// TIA Portal V17 export
// export: Created 2025-03-07T09:17:01.8029141Z, ExportSetting WithDefaults, DisplayName Totally Integrated Automation Portal, DisplayVersion V17 Update 8, DisplayName TIA Portal Openness, DisplayVersion V17 Update 8, DisplayName TIA Portal Version Control Interface, DisplayVersion V17, DisplayName SINAMICS Startdrive Advanced, DisplayVersion V17 SP2, DisplayName SINAMICS Startdrive G110M, G120, G120C, G120D, G120P, G115D, DisplayVersion V17 SP2, DisplayName SINAMICS Startdrive G130, G150, S120, S150, SINAMICS MV, S210, DisplayVersion V17 SP2, DisplayName STEP 7 Professional, DisplayVersion V17 Update 8, DisplayName SINUMERIK ONE STEP 7 Toolbox, DisplayVersion V17 Update 12, DisplayName SINUMERIK 840D sl STEP 7 Toolbox, DisplayVersion V17 Update 12, DisplayName STEP 7 Safety, DisplayVersion V17 Update 6, DisplayName WinCC Advanced, DisplayVersion V17 Update 8
FUNCTION "FC7341_POWDER_PLC_TO_MACHINE_INTERLOCK" : Void   // FC7341, LAD
{ S7_Optimized_Access := 'TRUE' }
VERSION : 0.1
// stored: AutoNumber false, IsIECCheckEnabled false, SetENOAutomatically false, UDAEnableTagReadback false
   VAR_TEMP
      COUNT_FOR_ERROR : Int;
      RET_VAL_1 : Int;
   END_VAR
   VAR CONSTANT
      FC_NUMBER : DInt := 7341;
   END_VAR
BEGIN

REGION Network 1: LIFE BIT
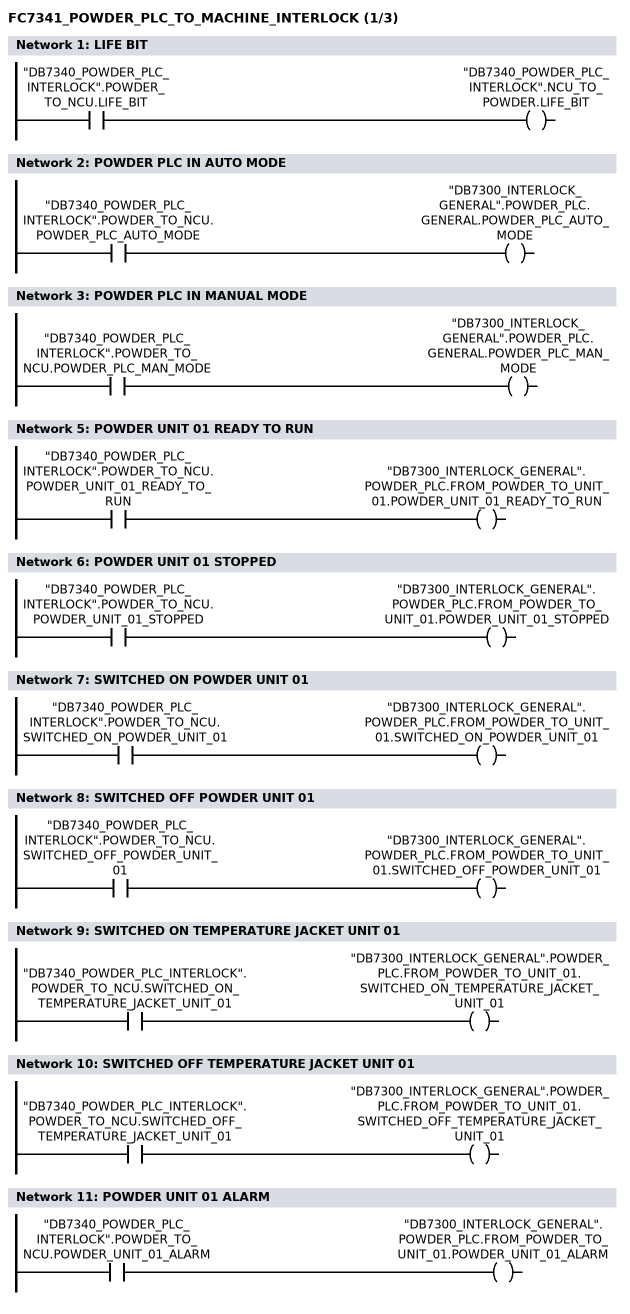
   RUNG wire#powerrail
      Contact( "DB7340_POWDER_PLC_INTERLOCK".POWDER_TO_NCU.LIFE_BIT )
      Coil( "DB7340_POWDER_PLC_INTERLOCK".NCU_TO_POWDER.LIFE_BIT )
   END_RUNG
   // the same network as SCL:
   "DB7340_POWDER_PLC_INTERLOCK".NCU_TO_POWDER.LIFE_BIT := "DB7340_POWDER_PLC_INTERLOCK".POWDER_TO_NCU.LIFE_BIT;
END_REGION

REGION Network 2: POWDER PLC IN AUTO MODE
   RUNG wire#powerrail
      Contact( "DB7340_POWDER_PLC_INTERLOCK".POWDER_TO_NCU.POWDER_PLC_AUTO_MODE )
      Coil( "DB7300_INTERLOCK_GENERAL".POWDER_PLC.GENERAL.POWDER_PLC_AUTO_MODE )
   END_RUNG
   // the same network as SCL:
   "DB7300_INTERLOCK_GENERAL".POWDER_PLC.GENERAL.POWDER_PLC_AUTO_MODE := "DB7340_POWDER_PLC_INTERLOCK".POWDER_TO_NCU.POWDER_PLC_AUTO_MODE;
END_REGION

REGION Network 3: POWDER PLC IN MANUAL MODE
   RUNG wire#powerrail
      Contact( "DB7340_POWDER_PLC_INTERLOCK".POWDER_TO_NCU.POWDER_PLC_MAN_MODE )
      Coil( "DB7300_INTERLOCK_GENERAL".POWDER_PLC.GENERAL.POWDER_PLC_MAN_MODE )
   END_RUNG
   // the same network as SCL:
   "DB7300_INTERLOCK_GENERAL".POWDER_PLC.GENERAL.POWDER_PLC_MAN_MODE := "DB7340_POWDER_PLC_INTERLOCK".POWDER_TO_NCU.POWDER_PLC_MAN_MODE;
END_REGION

REGION Network 4: //////////_UNIT_01_//////////
END_REGION

REGION Network 5: POWDER UNIT 01 READY TO RUN
   RUNG wire#powerrail
      Contact( "DB7340_POWDER_PLC_INTERLOCK".POWDER_TO_NCU.POWDER_UNIT_01_READY_TO_RUN )
      Coil( "DB7300_INTERLOCK_GENERAL".POWDER_PLC.FROM_POWDER_TO_UNIT_01.POWDER_UNIT_01_READY_TO_RUN )
   END_RUNG
   // the same network as SCL:
   "DB7300_INTERLOCK_GENERAL".POWDER_PLC.FROM_POWDER_TO_UNIT_01.POWDER_UNIT_01_READY_TO_RUN := "DB7340_POWDER_PLC_INTERLOCK".POWDER_TO_NCU.POWDER_UNIT_01_READY_TO_RUN;
END_REGION

REGION Network 6: POWDER UNIT 01 STOPPED
   RUNG wire#powerrail
      Contact( "DB7340_POWDER_PLC_INTERLOCK".POWDER_TO_NCU.POWDER_UNIT_01_STOPPED )
      Coil( "DB7300_INTERLOCK_GENERAL".POWDER_PLC.FROM_POWDER_TO_UNIT_01.POWDER_UNIT_01_STOPPED )
   END_RUNG
   // the same network as SCL:
   "DB7300_INTERLOCK_GENERAL".POWDER_PLC.FROM_POWDER_TO_UNIT_01.POWDER_UNIT_01_STOPPED := "DB7340_POWDER_PLC_INTERLOCK".POWDER_TO_NCU.POWDER_UNIT_01_STOPPED;
END_REGION

REGION Network 7: SWITCHED ON POWDER UNIT 01
   RUNG wire#powerrail
      Contact( "DB7340_POWDER_PLC_INTERLOCK".POWDER_TO_NCU.SWITCHED_ON_POWDER_UNIT_01 )
      Coil( "DB7300_INTERLOCK_GENERAL".POWDER_PLC.FROM_POWDER_TO_UNIT_01.SWITCHED_ON_POWDER_UNIT_01 )
   END_RUNG
   // the same network as SCL:
   "DB7300_INTERLOCK_GENERAL".POWDER_PLC.FROM_POWDER_TO_UNIT_01.SWITCHED_ON_POWDER_UNIT_01 := "DB7340_POWDER_PLC_INTERLOCK".POWDER_TO_NCU.SWITCHED_ON_POWDER_UNIT_01;
END_REGION

REGION Network 8: SWITCHED OFF POWDER UNIT 01
   RUNG wire#powerrail
      Contact( "DB7340_POWDER_PLC_INTERLOCK".POWDER_TO_NCU.SWITCHED_OFF_POWDER_UNIT_01 )
      Coil( "DB7300_INTERLOCK_GENERAL".POWDER_PLC.FROM_POWDER_TO_UNIT_01.SWITCHED_OFF_POWDER_UNIT_01 )
   END_RUNG
   // the same network as SCL:
   "DB7300_INTERLOCK_GENERAL".POWDER_PLC.FROM_POWDER_TO_UNIT_01.SWITCHED_OFF_POWDER_UNIT_01 := "DB7340_POWDER_PLC_INTERLOCK".POWDER_TO_NCU.SWITCHED_OFF_POWDER_UNIT_01;
END_REGION

REGION Network 9: SWITCHED ON TEMPERATURE JACKET UNIT 01
   RUNG wire#powerrail
      Contact( "DB7340_POWDER_PLC_INTERLOCK".POWDER_TO_NCU.SWITCHED_ON_TEMPERATURE_JACKET_UNIT_01 )
      Coil( "DB7300_INTERLOCK_GENERAL".POWDER_PLC.FROM_POWDER_TO_UNIT_01.SWITCHED_ON_TEMPERATURE_JACKET_UNIT_01 )
   END_RUNG
   // the same network as SCL:
   "DB7300_INTERLOCK_GENERAL".POWDER_PLC.FROM_POWDER_TO_UNIT_01.SWITCHED_ON_TEMPERATURE_JACKET_UNIT_01 := "DB7340_POWDER_PLC_INTERLOCK".POWDER_TO_NCU.SWITCHED_ON_TEMPERATURE_JACKET_UNIT_01;
END_REGION

REGION Network 10: SWITCHED OFF TEMPERATURE JACKET UNIT 01
   RUNG wire#powerrail
      Contact( "DB7340_POWDER_PLC_INTERLOCK".POWDER_TO_NCU.SWITCHED_OFF_TEMPERATURE_JACKET_UNIT_01 )
      Coil( "DB7300_INTERLOCK_GENERAL".POWDER_PLC.FROM_POWDER_TO_UNIT_01.SWITCHED_OFF_TEMPERATURE_JACKET_UNIT_01 )
   END_RUNG
   // the same network as SCL:
   "DB7300_INTERLOCK_GENERAL".POWDER_PLC.FROM_POWDER_TO_UNIT_01.SWITCHED_OFF_TEMPERATURE_JACKET_UNIT_01 := "DB7340_POWDER_PLC_INTERLOCK".POWDER_TO_NCU.SWITCHED_OFF_TEMPERATURE_JACKET_UNIT_01;
END_REGION

REGION Network 11: POWDER UNIT 01 ALARM
   RUNG wire#powerrail
      Contact( "DB7340_POWDER_PLC_INTERLOCK".POWDER_TO_NCU.POWDER_UNIT_01_ALARM )
      Coil( "DB7300_INTERLOCK_GENERAL".POWDER_PLC.FROM_POWDER_TO_UNIT_01.POWDER_UNIT_01_ALARM )
   END_RUNG
   // the same network as SCL:
   "DB7300_INTERLOCK_GENERAL".POWDER_PLC.FROM_POWDER_TO_UNIT_01.POWDER_UNIT_01_ALARM := "DB7340_POWDER_PLC_INTERLOCK".POWDER_TO_NCU.POWDER_UNIT_01_ALARM;
END_REGION

REGION Network 12: POWDER FEEDER 1 ACTUAL VALUES
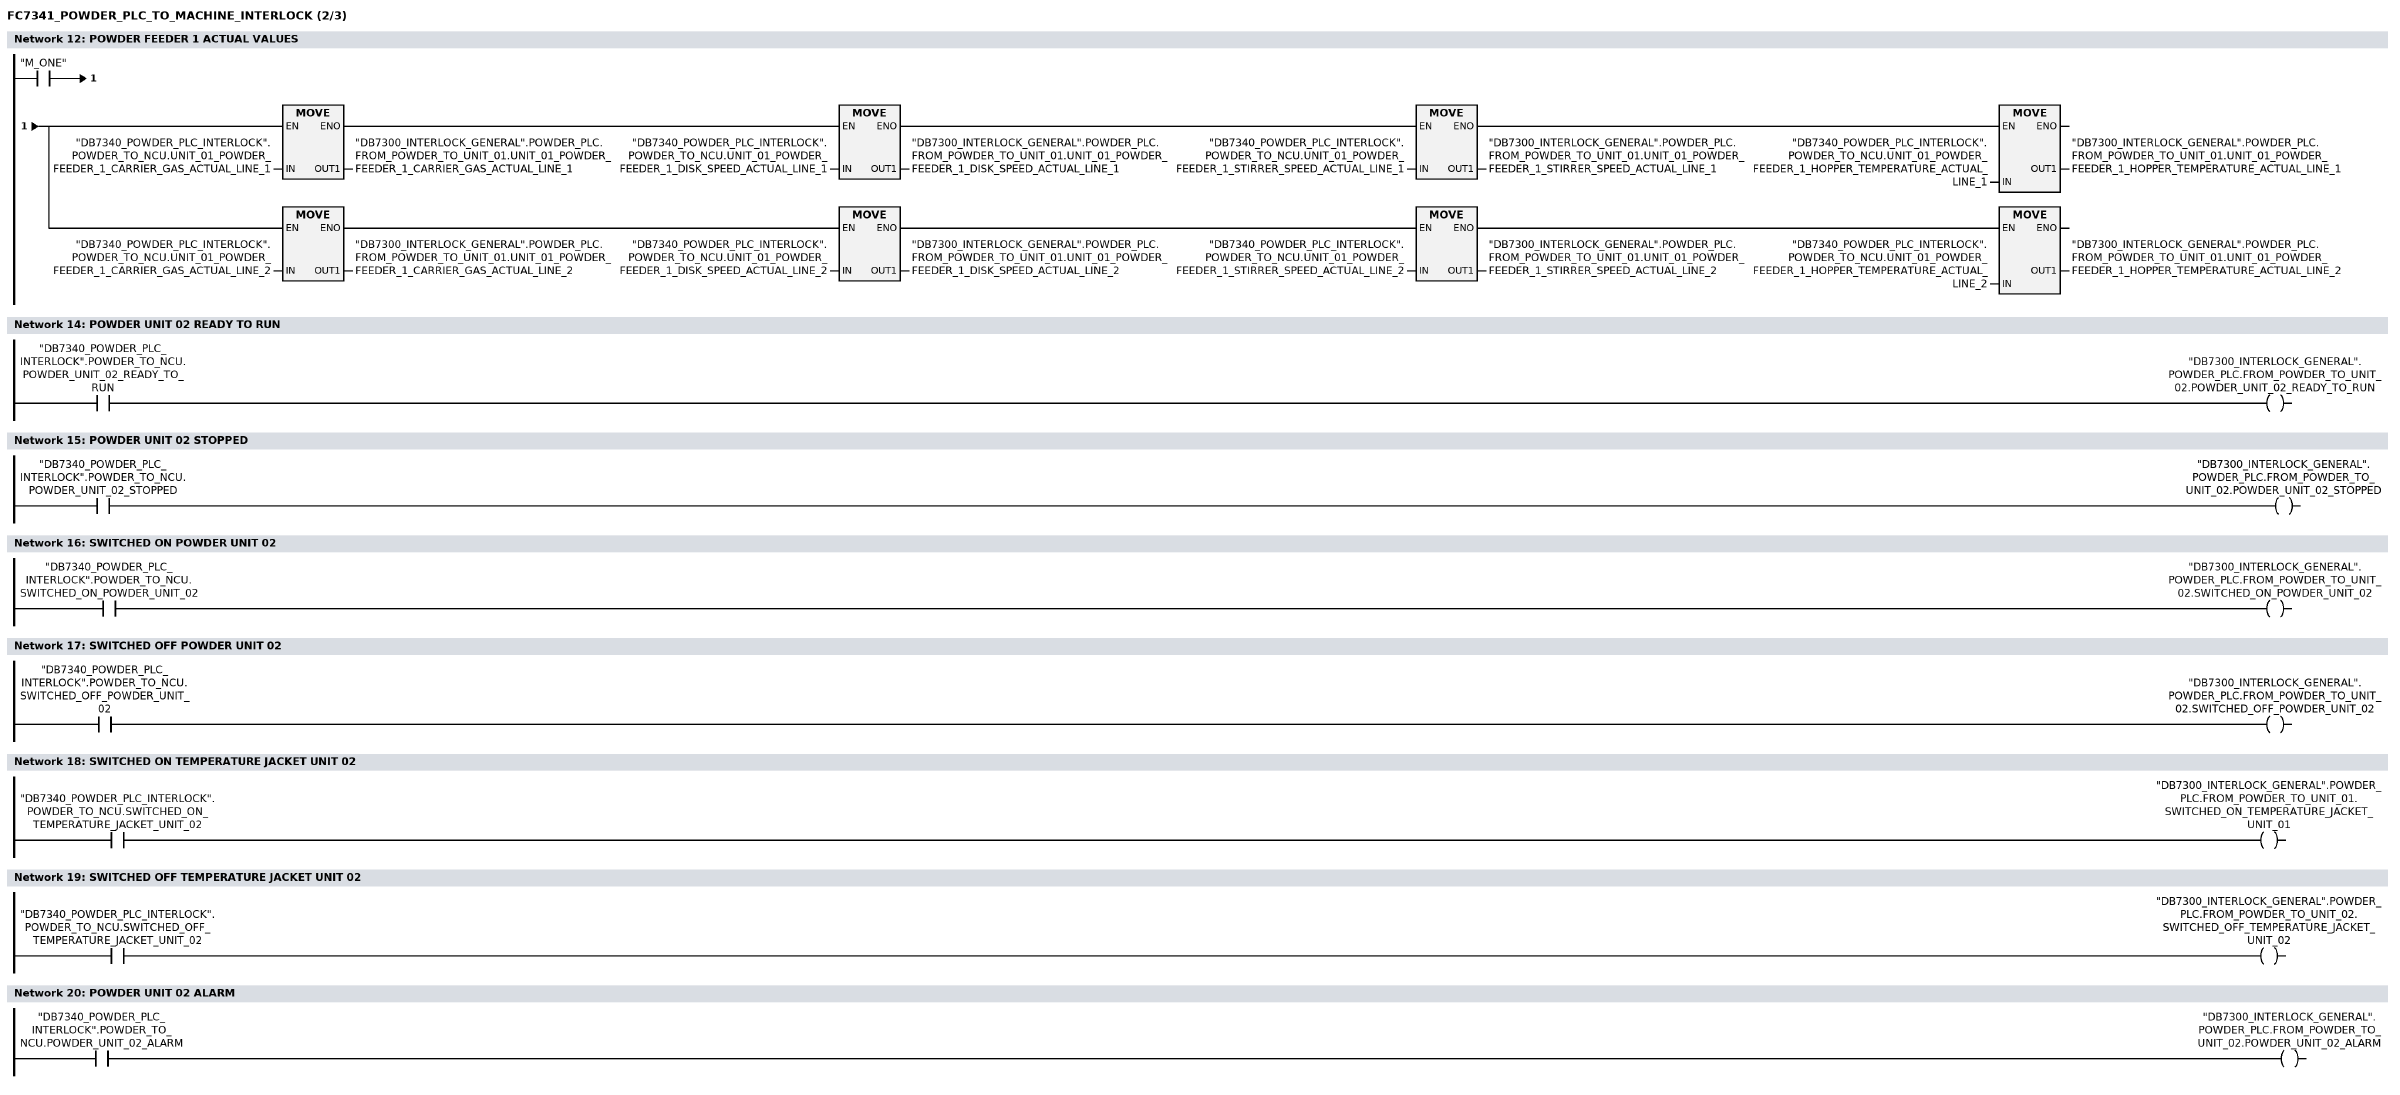
   RUNG wire#powerrail
      Contact( "M_ONE" )
      wire#w1
      Move(in := "DB7340_POWDER_PLC_INTERLOCK".POWDER_TO_NCU.UNIT_01_POWDER_FEEDER_1_CARRIER_GAS_ACTUAL_LINE_1, out1 => "DB7300_INTERLOCK_GENERAL".POWDER_PLC.FROM_POWDER_TO_UNIT_01.UNIT_01_POWDER_FEEDER_1_CARRIER_GAS_ACTUAL_LINE_1)
      Move(in := "DB7340_POWDER_PLC_INTERLOCK".POWDER_TO_NCU.UNIT_01_POWDER_FEEDER_1_DISK_SPEED_ACTUAL_LINE_1, out1 => "DB7300_INTERLOCK_GENERAL".POWDER_PLC.FROM_POWDER_TO_UNIT_01.UNIT_01_POWDER_FEEDER_1_DISK_SPEED_ACTUAL_LINE_1)
      Move(in := "DB7340_POWDER_PLC_INTERLOCK".POWDER_TO_NCU.UNIT_01_POWDER_FEEDER_1_STIRRER_SPEED_ACTUAL_LINE_1, out1 => "DB7300_INTERLOCK_GENERAL".POWDER_PLC.FROM_POWDER_TO_UNIT_01.UNIT_01_POWDER_FEEDER_1_STIRRER_SPEED_ACTUAL_LINE_1)
      Move(in := "DB7340_POWDER_PLC_INTERLOCK".POWDER_TO_NCU.UNIT_01_POWDER_FEEDER_1_HOPPER_TEMPERATURE_ACTUAL_LINE_1, out1 => "DB7300_INTERLOCK_GENERAL".POWDER_PLC.FROM_POWDER_TO_UNIT_01.UNIT_01_POWDER_FEEDER_1_HOPPER_TEMPERATURE_ACTUAL_LINE_1)
   END_RUNG
   RUNG wire#w1
      Move(in := "DB7340_POWDER_PLC_INTERLOCK".POWDER_TO_NCU.UNIT_01_POWDER_FEEDER_1_CARRIER_GAS_ACTUAL_LINE_2, out1 => "DB7300_INTERLOCK_GENERAL".POWDER_PLC.FROM_POWDER_TO_UNIT_01.UNIT_01_POWDER_FEEDER_1_CARRIER_GAS_ACTUAL_LINE_2)
      Move(in := "DB7340_POWDER_PLC_INTERLOCK".POWDER_TO_NCU.UNIT_01_POWDER_FEEDER_1_DISK_SPEED_ACTUAL_LINE_2, out1 => "DB7300_INTERLOCK_GENERAL".POWDER_PLC.FROM_POWDER_TO_UNIT_01.UNIT_01_POWDER_FEEDER_1_DISK_SPEED_ACTUAL_LINE_2)
      Move(in := "DB7340_POWDER_PLC_INTERLOCK".POWDER_TO_NCU.UNIT_01_POWDER_FEEDER_1_STIRRER_SPEED_ACTUAL_LINE_2, out1 => "DB7300_INTERLOCK_GENERAL".POWDER_PLC.FROM_POWDER_TO_UNIT_01.UNIT_01_POWDER_FEEDER_1_STIRRER_SPEED_ACTUAL_LINE_2)
      Move(in := "DB7340_POWDER_PLC_INTERLOCK".POWDER_TO_NCU.UNIT_01_POWDER_FEEDER_1_HOPPER_TEMPERATURE_ACTUAL_LINE_2, out1 => "DB7300_INTERLOCK_GENERAL".POWDER_PLC.FROM_POWDER_TO_UNIT_01.UNIT_01_POWDER_FEEDER_1_HOPPER_TEMPERATURE_ACTUAL_LINE_2)
   END_RUNG
   // the same network as SCL:
   IF "M_ONE" THEN
       "DB7300_INTERLOCK_GENERAL".POWDER_PLC.FROM_POWDER_TO_UNIT_01.UNIT_01_POWDER_FEEDER_1_CARRIER_GAS_ACTUAL_LINE_1 := "DB7340_POWDER_PLC_INTERLOCK".POWDER_TO_NCU.UNIT_01_POWDER_FEEDER_1_CARRIER_GAS_ACTUAL_LINE_1;
       "DB7300_INTERLOCK_GENERAL".POWDER_PLC.FROM_POWDER_TO_UNIT_01.UNIT_01_POWDER_FEEDER_1_DISK_SPEED_ACTUAL_LINE_1 := "DB7340_POWDER_PLC_INTERLOCK".POWDER_TO_NCU.UNIT_01_POWDER_FEEDER_1_DISK_SPEED_ACTUAL_LINE_1;
       "DB7300_INTERLOCK_GENERAL".POWDER_PLC.FROM_POWDER_TO_UNIT_01.UNIT_01_POWDER_FEEDER_1_STIRRER_SPEED_ACTUAL_LINE_1 := "DB7340_POWDER_PLC_INTERLOCK".POWDER_TO_NCU.UNIT_01_POWDER_FEEDER_1_STIRRER_SPEED_ACTUAL_LINE_1;
       "DB7300_INTERLOCK_GENERAL".POWDER_PLC.FROM_POWDER_TO_UNIT_01.UNIT_01_POWDER_FEEDER_1_HOPPER_TEMPERATURE_ACTUAL_LINE_1 := "DB7340_POWDER_PLC_INTERLOCK".POWDER_TO_NCU.UNIT_01_POWDER_FEEDER_1_HOPPER_TEMPERATURE_ACTUAL_LINE_1;
       "DB7300_INTERLOCK_GENERAL".POWDER_PLC.FROM_POWDER_TO_UNIT_01.UNIT_01_POWDER_FEEDER_1_CARRIER_GAS_ACTUAL_LINE_2 := "DB7340_POWDER_PLC_INTERLOCK".POWDER_TO_NCU.UNIT_01_POWDER_FEEDER_1_CARRIER_GAS_ACTUAL_LINE_2;
       "DB7300_INTERLOCK_GENERAL".POWDER_PLC.FROM_POWDER_TO_UNIT_01.UNIT_01_POWDER_FEEDER_1_DISK_SPEED_ACTUAL_LINE_2 := "DB7340_POWDER_PLC_INTERLOCK".POWDER_TO_NCU.UNIT_01_POWDER_FEEDER_1_DISK_SPEED_ACTUAL_LINE_2;
       "DB7300_INTERLOCK_GENERAL".POWDER_PLC.FROM_POWDER_TO_UNIT_01.UNIT_01_POWDER_FEEDER_1_STIRRER_SPEED_ACTUAL_LINE_2 := "DB7340_POWDER_PLC_INTERLOCK".POWDER_TO_NCU.UNIT_01_POWDER_FEEDER_1_STIRRER_SPEED_ACTUAL_LINE_2;
       "DB7300_INTERLOCK_GENERAL".POWDER_PLC.FROM_POWDER_TO_UNIT_01.UNIT_01_POWDER_FEEDER_1_HOPPER_TEMPERATURE_ACTUAL_LINE_2 := "DB7340_POWDER_PLC_INTERLOCK".POWDER_TO_NCU.UNIT_01_POWDER_FEEDER_1_HOPPER_TEMPERATURE_ACTUAL_LINE_2;
   END_IF;
END_REGION

REGION Network 13: //////////_UNIT_02_//////////
END_REGION

REGION Network 14: POWDER UNIT 02 READY TO RUN
   RUNG wire#powerrail
      Contact( "DB7340_POWDER_PLC_INTERLOCK".POWDER_TO_NCU.POWDER_UNIT_02_READY_TO_RUN )
      Coil( "DB7300_INTERLOCK_GENERAL".POWDER_PLC.FROM_POWDER_TO_UNIT_02.POWDER_UNIT_02_READY_TO_RUN )
   END_RUNG
   // the same network as SCL:
   "DB7300_INTERLOCK_GENERAL".POWDER_PLC.FROM_POWDER_TO_UNIT_02.POWDER_UNIT_02_READY_TO_RUN := "DB7340_POWDER_PLC_INTERLOCK".POWDER_TO_NCU.POWDER_UNIT_02_READY_TO_RUN;
END_REGION

REGION Network 15: POWDER UNIT 02 STOPPED
   RUNG wire#powerrail
      Contact( "DB7340_POWDER_PLC_INTERLOCK".POWDER_TO_NCU.POWDER_UNIT_02_STOPPED )
      Coil( "DB7300_INTERLOCK_GENERAL".POWDER_PLC.FROM_POWDER_TO_UNIT_02.POWDER_UNIT_02_STOPPED )
   END_RUNG
   // the same network as SCL:
   "DB7300_INTERLOCK_GENERAL".POWDER_PLC.FROM_POWDER_TO_UNIT_02.POWDER_UNIT_02_STOPPED := "DB7340_POWDER_PLC_INTERLOCK".POWDER_TO_NCU.POWDER_UNIT_02_STOPPED;
END_REGION

REGION Network 16: SWITCHED ON POWDER UNIT 02
   RUNG wire#powerrail
      Contact( "DB7340_POWDER_PLC_INTERLOCK".POWDER_TO_NCU.SWITCHED_ON_POWDER_UNIT_02 )
      Coil( "DB7300_INTERLOCK_GENERAL".POWDER_PLC.FROM_POWDER_TO_UNIT_02.SWITCHED_ON_POWDER_UNIT_02 )
   END_RUNG
   // the same network as SCL:
   "DB7300_INTERLOCK_GENERAL".POWDER_PLC.FROM_POWDER_TO_UNIT_02.SWITCHED_ON_POWDER_UNIT_02 := "DB7340_POWDER_PLC_INTERLOCK".POWDER_TO_NCU.SWITCHED_ON_POWDER_UNIT_02;
END_REGION

REGION Network 17: SWITCHED OFF POWDER UNIT 02
   RUNG wire#powerrail
      Contact( "DB7340_POWDER_PLC_INTERLOCK".POWDER_TO_NCU.SWITCHED_OFF_POWDER_UNIT_02 )
      Coil( "DB7300_INTERLOCK_GENERAL".POWDER_PLC.FROM_POWDER_TO_UNIT_02.SWITCHED_OFF_POWDER_UNIT_02 )
   END_RUNG
   // the same network as SCL:
   "DB7300_INTERLOCK_GENERAL".POWDER_PLC.FROM_POWDER_TO_UNIT_02.SWITCHED_OFF_POWDER_UNIT_02 := "DB7340_POWDER_PLC_INTERLOCK".POWDER_TO_NCU.SWITCHED_OFF_POWDER_UNIT_02;
END_REGION

REGION Network 18: SWITCHED ON TEMPERATURE JACKET UNIT 02
   RUNG wire#powerrail
      Contact( "DB7340_POWDER_PLC_INTERLOCK".POWDER_TO_NCU.SWITCHED_ON_TEMPERATURE_JACKET_UNIT_02 )
      Coil( "DB7300_INTERLOCK_GENERAL".POWDER_PLC.FROM_POWDER_TO_UNIT_01.SWITCHED_ON_TEMPERATURE_JACKET_UNIT_01 )
   END_RUNG
   // the same network as SCL:
   "DB7300_INTERLOCK_GENERAL".POWDER_PLC.FROM_POWDER_TO_UNIT_01.SWITCHED_ON_TEMPERATURE_JACKET_UNIT_01 := "DB7340_POWDER_PLC_INTERLOCK".POWDER_TO_NCU.SWITCHED_ON_TEMPERATURE_JACKET_UNIT_02;
END_REGION

REGION Network 19: SWITCHED OFF TEMPERATURE JACKET UNIT 02
   RUNG wire#powerrail
      Contact( "DB7340_POWDER_PLC_INTERLOCK".POWDER_TO_NCU.SWITCHED_OFF_TEMPERATURE_JACKET_UNIT_02 )
      Coil( "DB7300_INTERLOCK_GENERAL".POWDER_PLC.FROM_POWDER_TO_UNIT_02.SWITCHED_OFF_TEMPERATURE_JACKET_UNIT_02 )
   END_RUNG
   // the same network as SCL:
   "DB7300_INTERLOCK_GENERAL".POWDER_PLC.FROM_POWDER_TO_UNIT_02.SWITCHED_OFF_TEMPERATURE_JACKET_UNIT_02 := "DB7340_POWDER_PLC_INTERLOCK".POWDER_TO_NCU.SWITCHED_OFF_TEMPERATURE_JACKET_UNIT_02;
END_REGION

REGION Network 20: POWDER UNIT 02 ALARM
   RUNG wire#powerrail
      Contact( "DB7340_POWDER_PLC_INTERLOCK".POWDER_TO_NCU.POWDER_UNIT_02_ALARM )
      Coil( "DB7300_INTERLOCK_GENERAL".POWDER_PLC.FROM_POWDER_TO_UNIT_02.POWDER_UNIT_02_ALARM )
   END_RUNG
   // the same network as SCL:
   "DB7300_INTERLOCK_GENERAL".POWDER_PLC.FROM_POWDER_TO_UNIT_02.POWDER_UNIT_02_ALARM := "DB7340_POWDER_PLC_INTERLOCK".POWDER_TO_NCU.POWDER_UNIT_02_ALARM;
END_REGION

REGION Network 21: POWDER FEEDER 1 ACTUAL VALUES
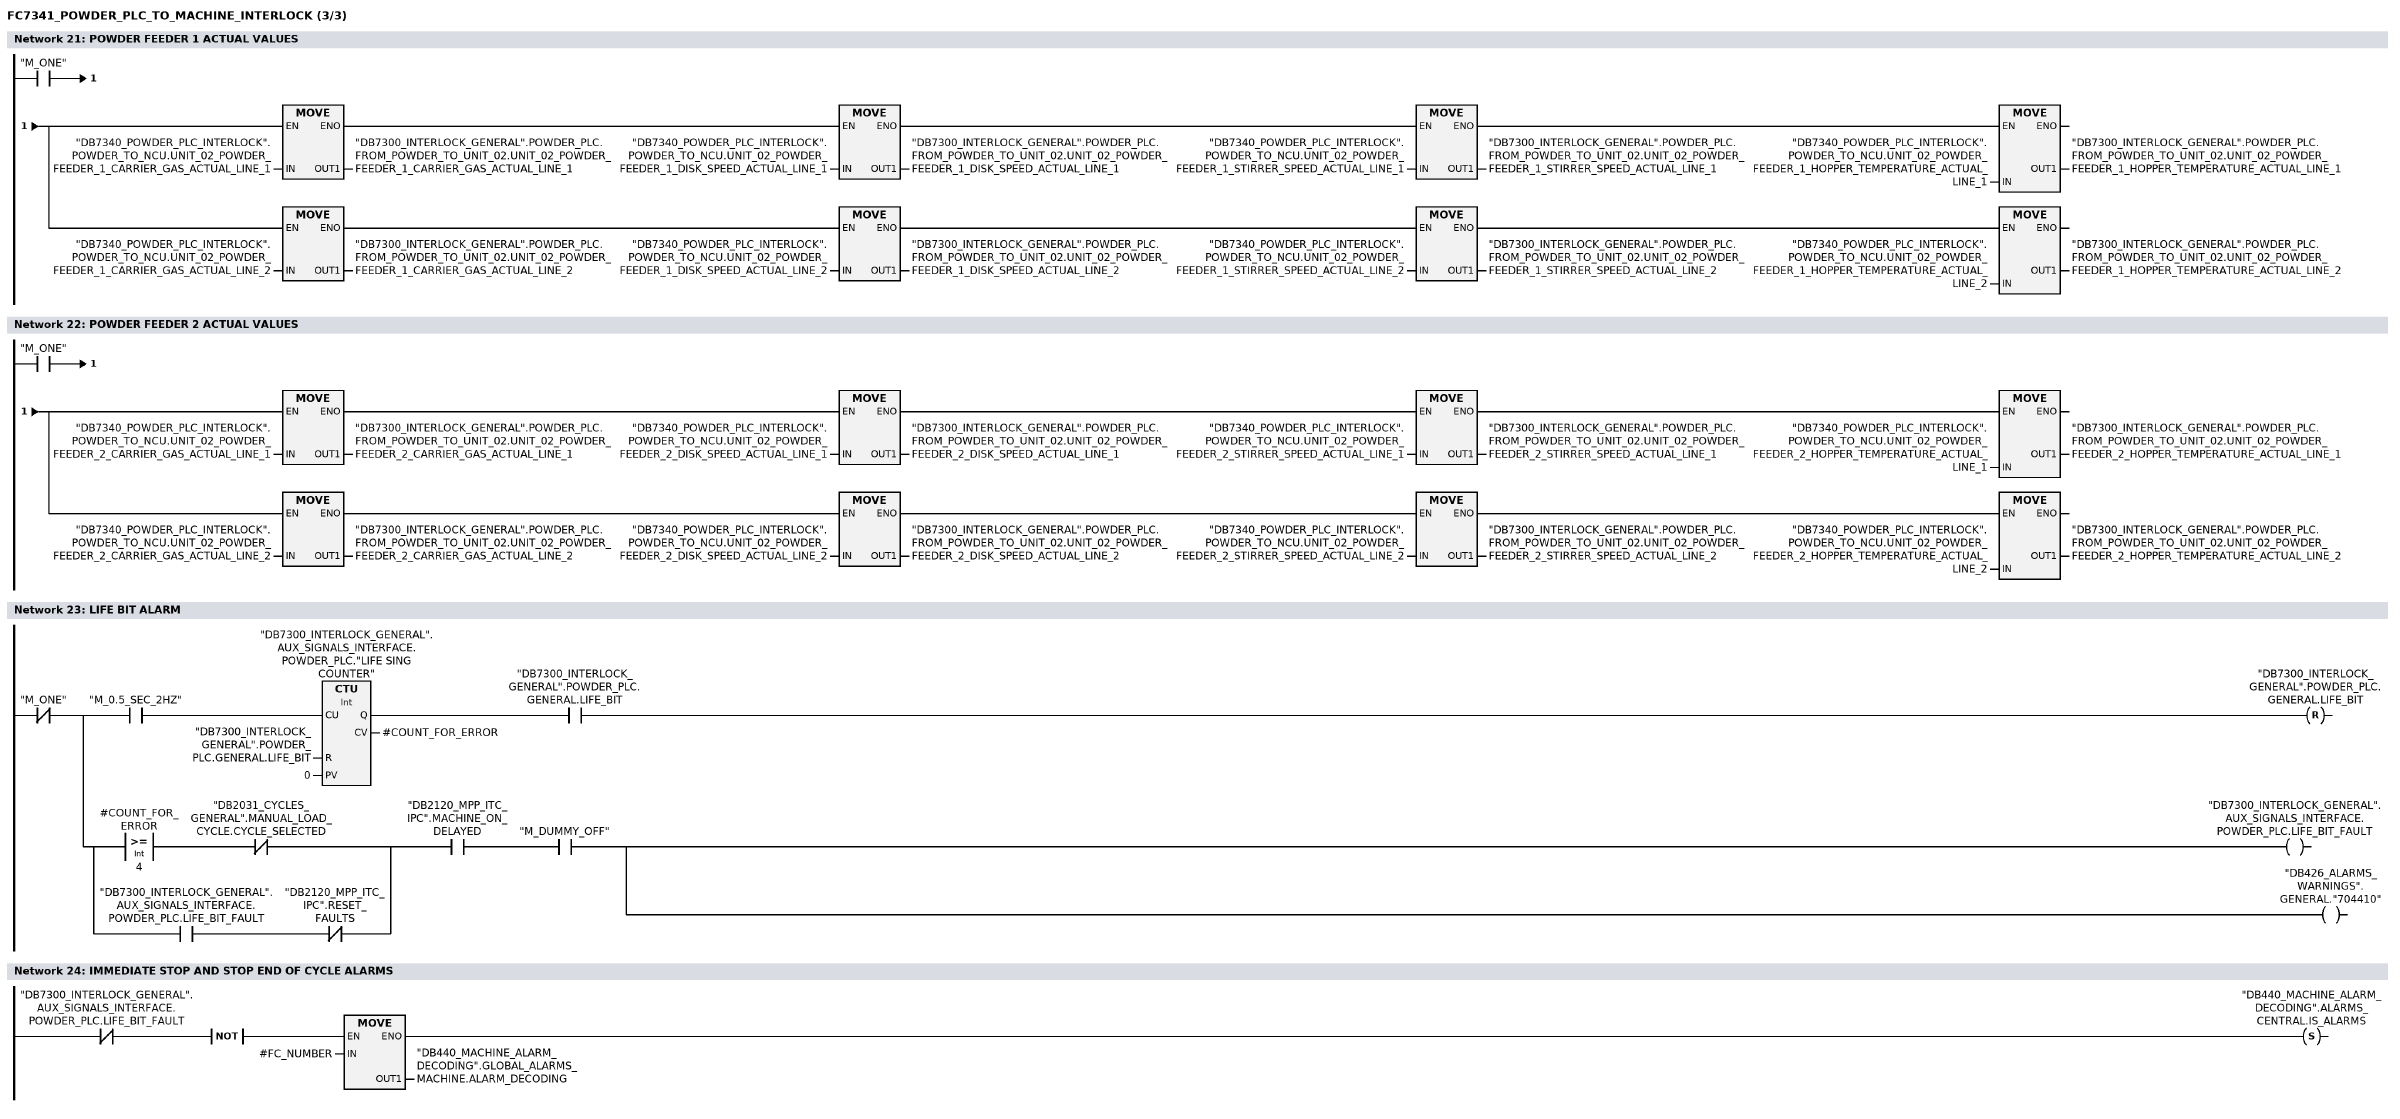
   RUNG wire#powerrail
      Contact( "M_ONE" )
      wire#w1
      Move(in := "DB7340_POWDER_PLC_INTERLOCK".POWDER_TO_NCU.UNIT_02_POWDER_FEEDER_1_CARRIER_GAS_ACTUAL_LINE_1, out1 => "DB7300_INTERLOCK_GENERAL".POWDER_PLC.FROM_POWDER_TO_UNIT_02.UNIT_02_POWDER_FEEDER_1_CARRIER_GAS_ACTUAL_LINE_1)
      Move(in := "DB7340_POWDER_PLC_INTERLOCK".POWDER_TO_NCU.UNIT_02_POWDER_FEEDER_1_DISK_SPEED_ACTUAL_LINE_1, out1 => "DB7300_INTERLOCK_GENERAL".POWDER_PLC.FROM_POWDER_TO_UNIT_02.UNIT_02_POWDER_FEEDER_1_DISK_SPEED_ACTUAL_LINE_1)
      Move(in := "DB7340_POWDER_PLC_INTERLOCK".POWDER_TO_NCU.UNIT_02_POWDER_FEEDER_1_STIRRER_SPEED_ACTUAL_LINE_1, out1 => "DB7300_INTERLOCK_GENERAL".POWDER_PLC.FROM_POWDER_TO_UNIT_02.UNIT_02_POWDER_FEEDER_1_STIRRER_SPEED_ACTUAL_LINE_1)
      Move(in := "DB7340_POWDER_PLC_INTERLOCK".POWDER_TO_NCU.UNIT_02_POWDER_FEEDER_1_HOPPER_TEMPERATURE_ACTUAL_LINE_1, out1 => "DB7300_INTERLOCK_GENERAL".POWDER_PLC.FROM_POWDER_TO_UNIT_02.UNIT_02_POWDER_FEEDER_1_HOPPER_TEMPERATURE_ACTUAL_LINE_1)
   END_RUNG
   RUNG wire#w1
      Move(in := "DB7340_POWDER_PLC_INTERLOCK".POWDER_TO_NCU.UNIT_02_POWDER_FEEDER_1_CARRIER_GAS_ACTUAL_LINE_2, out1 => "DB7300_INTERLOCK_GENERAL".POWDER_PLC.FROM_POWDER_TO_UNIT_02.UNIT_02_POWDER_FEEDER_1_CARRIER_GAS_ACTUAL_LINE_2)
      Move(in := "DB7340_POWDER_PLC_INTERLOCK".POWDER_TO_NCU.UNIT_02_POWDER_FEEDER_1_DISK_SPEED_ACTUAL_LINE_2, out1 => "DB7300_INTERLOCK_GENERAL".POWDER_PLC.FROM_POWDER_TO_UNIT_02.UNIT_02_POWDER_FEEDER_1_DISK_SPEED_ACTUAL_LINE_2)
      Move(in := "DB7340_POWDER_PLC_INTERLOCK".POWDER_TO_NCU.UNIT_02_POWDER_FEEDER_1_STIRRER_SPEED_ACTUAL_LINE_2, out1 => "DB7300_INTERLOCK_GENERAL".POWDER_PLC.FROM_POWDER_TO_UNIT_02.UNIT_02_POWDER_FEEDER_1_STIRRER_SPEED_ACTUAL_LINE_2)
      Move(in := "DB7340_POWDER_PLC_INTERLOCK".POWDER_TO_NCU.UNIT_02_POWDER_FEEDER_1_HOPPER_TEMPERATURE_ACTUAL_LINE_2, out1 => "DB7300_INTERLOCK_GENERAL".POWDER_PLC.FROM_POWDER_TO_UNIT_02.UNIT_02_POWDER_FEEDER_1_HOPPER_TEMPERATURE_ACTUAL_LINE_2)
   END_RUNG
   // the same network as SCL:
   IF "M_ONE" THEN
       "DB7300_INTERLOCK_GENERAL".POWDER_PLC.FROM_POWDER_TO_UNIT_02.UNIT_02_POWDER_FEEDER_1_CARRIER_GAS_ACTUAL_LINE_1 := "DB7340_POWDER_PLC_INTERLOCK".POWDER_TO_NCU.UNIT_02_POWDER_FEEDER_1_CARRIER_GAS_ACTUAL_LINE_1;
       "DB7300_INTERLOCK_GENERAL".POWDER_PLC.FROM_POWDER_TO_UNIT_02.UNIT_02_POWDER_FEEDER_1_DISK_SPEED_ACTUAL_LINE_1 := "DB7340_POWDER_PLC_INTERLOCK".POWDER_TO_NCU.UNIT_02_POWDER_FEEDER_1_DISK_SPEED_ACTUAL_LINE_1;
       "DB7300_INTERLOCK_GENERAL".POWDER_PLC.FROM_POWDER_TO_UNIT_02.UNIT_02_POWDER_FEEDER_1_STIRRER_SPEED_ACTUAL_LINE_1 := "DB7340_POWDER_PLC_INTERLOCK".POWDER_TO_NCU.UNIT_02_POWDER_FEEDER_1_STIRRER_SPEED_ACTUAL_LINE_1;
       "DB7300_INTERLOCK_GENERAL".POWDER_PLC.FROM_POWDER_TO_UNIT_02.UNIT_02_POWDER_FEEDER_1_HOPPER_TEMPERATURE_ACTUAL_LINE_1 := "DB7340_POWDER_PLC_INTERLOCK".POWDER_TO_NCU.UNIT_02_POWDER_FEEDER_1_HOPPER_TEMPERATURE_ACTUAL_LINE_1;
       "DB7300_INTERLOCK_GENERAL".POWDER_PLC.FROM_POWDER_TO_UNIT_02.UNIT_02_POWDER_FEEDER_1_CARRIER_GAS_ACTUAL_LINE_2 := "DB7340_POWDER_PLC_INTERLOCK".POWDER_TO_NCU.UNIT_02_POWDER_FEEDER_1_CARRIER_GAS_ACTUAL_LINE_2;
       "DB7300_INTERLOCK_GENERAL".POWDER_PLC.FROM_POWDER_TO_UNIT_02.UNIT_02_POWDER_FEEDER_1_DISK_SPEED_ACTUAL_LINE_2 := "DB7340_POWDER_PLC_INTERLOCK".POWDER_TO_NCU.UNIT_02_POWDER_FEEDER_1_DISK_SPEED_ACTUAL_LINE_2;
       "DB7300_INTERLOCK_GENERAL".POWDER_PLC.FROM_POWDER_TO_UNIT_02.UNIT_02_POWDER_FEEDER_1_STIRRER_SPEED_ACTUAL_LINE_2 := "DB7340_POWDER_PLC_INTERLOCK".POWDER_TO_NCU.UNIT_02_POWDER_FEEDER_1_STIRRER_SPEED_ACTUAL_LINE_2;
       "DB7300_INTERLOCK_GENERAL".POWDER_PLC.FROM_POWDER_TO_UNIT_02.UNIT_02_POWDER_FEEDER_1_HOPPER_TEMPERATURE_ACTUAL_LINE_2 := "DB7340_POWDER_PLC_INTERLOCK".POWDER_TO_NCU.UNIT_02_POWDER_FEEDER_1_HOPPER_TEMPERATURE_ACTUAL_LINE_2;
   END_IF;
END_REGION

REGION Network 22: POWDER FEEDER 2 ACTUAL VALUES
   RUNG wire#powerrail
      Contact( "M_ONE" )
      wire#w1
      Move(in := "DB7340_POWDER_PLC_INTERLOCK".POWDER_TO_NCU.UNIT_02_POWDER_FEEDER_2_CARRIER_GAS_ACTUAL_LINE_1, out1 => "DB7300_INTERLOCK_GENERAL".POWDER_PLC.FROM_POWDER_TO_UNIT_02.UNIT_02_POWDER_FEEDER_2_CARRIER_GAS_ACTUAL_LINE_1)
      Move(in := "DB7340_POWDER_PLC_INTERLOCK".POWDER_TO_NCU.UNIT_02_POWDER_FEEDER_2_DISK_SPEED_ACTUAL_LINE_1, out1 => "DB7300_INTERLOCK_GENERAL".POWDER_PLC.FROM_POWDER_TO_UNIT_02.UNIT_02_POWDER_FEEDER_2_DISK_SPEED_ACTUAL_LINE_1)
      Move(in := "DB7340_POWDER_PLC_INTERLOCK".POWDER_TO_NCU.UNIT_02_POWDER_FEEDER_2_STIRRER_SPEED_ACTUAL_LINE_1, out1 => "DB7300_INTERLOCK_GENERAL".POWDER_PLC.FROM_POWDER_TO_UNIT_02.UNIT_02_POWDER_FEEDER_2_STIRRER_SPEED_ACTUAL_LINE_1)
      Move(in := "DB7340_POWDER_PLC_INTERLOCK".POWDER_TO_NCU.UNIT_02_POWDER_FEEDER_2_HOPPER_TEMPERATURE_ACTUAL_LINE_1, out1 => "DB7300_INTERLOCK_GENERAL".POWDER_PLC.FROM_POWDER_TO_UNIT_02.UNIT_02_POWDER_FEEDER_2_HOPPER_TEMPERATURE_ACTUAL_LINE_1)
   END_RUNG
   RUNG wire#w1
      Move(in := "DB7340_POWDER_PLC_INTERLOCK".POWDER_TO_NCU.UNIT_02_POWDER_FEEDER_2_CARRIER_GAS_ACTUAL_LINE_2, out1 => "DB7300_INTERLOCK_GENERAL".POWDER_PLC.FROM_POWDER_TO_UNIT_02.UNIT_02_POWDER_FEEDER_2_CARRIER_GAS_ACTUAL_LINE_2)
      Move(in := "DB7340_POWDER_PLC_INTERLOCK".POWDER_TO_NCU.UNIT_02_POWDER_FEEDER_2_DISK_SPEED_ACTUAL_LINE_2, out1 => "DB7300_INTERLOCK_GENERAL".POWDER_PLC.FROM_POWDER_TO_UNIT_02.UNIT_02_POWDER_FEEDER_2_DISK_SPEED_ACTUAL_LINE_2)
      Move(in := "DB7340_POWDER_PLC_INTERLOCK".POWDER_TO_NCU.UNIT_02_POWDER_FEEDER_2_STIRRER_SPEED_ACTUAL_LINE_2, out1 => "DB7300_INTERLOCK_GENERAL".POWDER_PLC.FROM_POWDER_TO_UNIT_02.UNIT_02_POWDER_FEEDER_2_STIRRER_SPEED_ACTUAL_LINE_2)
      Move(in := "DB7340_POWDER_PLC_INTERLOCK".POWDER_TO_NCU.UNIT_02_POWDER_FEEDER_2_HOPPER_TEMPERATURE_ACTUAL_LINE_2, out1 => "DB7300_INTERLOCK_GENERAL".POWDER_PLC.FROM_POWDER_TO_UNIT_02.UNIT_02_POWDER_FEEDER_2_HOPPER_TEMPERATURE_ACTUAL_LINE_2)
   END_RUNG
   // the same network as SCL:
   IF "M_ONE" THEN
       "DB7300_INTERLOCK_GENERAL".POWDER_PLC.FROM_POWDER_TO_UNIT_02.UNIT_02_POWDER_FEEDER_2_CARRIER_GAS_ACTUAL_LINE_1 := "DB7340_POWDER_PLC_INTERLOCK".POWDER_TO_NCU.UNIT_02_POWDER_FEEDER_2_CARRIER_GAS_ACTUAL_LINE_1;
       "DB7300_INTERLOCK_GENERAL".POWDER_PLC.FROM_POWDER_TO_UNIT_02.UNIT_02_POWDER_FEEDER_2_DISK_SPEED_ACTUAL_LINE_1 := "DB7340_POWDER_PLC_INTERLOCK".POWDER_TO_NCU.UNIT_02_POWDER_FEEDER_2_DISK_SPEED_ACTUAL_LINE_1;
       "DB7300_INTERLOCK_GENERAL".POWDER_PLC.FROM_POWDER_TO_UNIT_02.UNIT_02_POWDER_FEEDER_2_STIRRER_SPEED_ACTUAL_LINE_1 := "DB7340_POWDER_PLC_INTERLOCK".POWDER_TO_NCU.UNIT_02_POWDER_FEEDER_2_STIRRER_SPEED_ACTUAL_LINE_1;
       "DB7300_INTERLOCK_GENERAL".POWDER_PLC.FROM_POWDER_TO_UNIT_02.UNIT_02_POWDER_FEEDER_2_HOPPER_TEMPERATURE_ACTUAL_LINE_1 := "DB7340_POWDER_PLC_INTERLOCK".POWDER_TO_NCU.UNIT_02_POWDER_FEEDER_2_HOPPER_TEMPERATURE_ACTUAL_LINE_1;
       "DB7300_INTERLOCK_GENERAL".POWDER_PLC.FROM_POWDER_TO_UNIT_02.UNIT_02_POWDER_FEEDER_2_CARRIER_GAS_ACTUAL_LINE_2 := "DB7340_POWDER_PLC_INTERLOCK".POWDER_TO_NCU.UNIT_02_POWDER_FEEDER_2_CARRIER_GAS_ACTUAL_LINE_2;
       "DB7300_INTERLOCK_GENERAL".POWDER_PLC.FROM_POWDER_TO_UNIT_02.UNIT_02_POWDER_FEEDER_2_DISK_SPEED_ACTUAL_LINE_2 := "DB7340_POWDER_PLC_INTERLOCK".POWDER_TO_NCU.UNIT_02_POWDER_FEEDER_2_DISK_SPEED_ACTUAL_LINE_2;
       "DB7300_INTERLOCK_GENERAL".POWDER_PLC.FROM_POWDER_TO_UNIT_02.UNIT_02_POWDER_FEEDER_2_STIRRER_SPEED_ACTUAL_LINE_2 := "DB7340_POWDER_PLC_INTERLOCK".POWDER_TO_NCU.UNIT_02_POWDER_FEEDER_2_STIRRER_SPEED_ACTUAL_LINE_2;
       "DB7300_INTERLOCK_GENERAL".POWDER_PLC.FROM_POWDER_TO_UNIT_02.UNIT_02_POWDER_FEEDER_2_HOPPER_TEMPERATURE_ACTUAL_LINE_2 := "DB7340_POWDER_PLC_INTERLOCK".POWDER_TO_NCU.UNIT_02_POWDER_FEEDER_2_HOPPER_TEMPERATURE_ACTUAL_LINE_2;
   END_IF;
END_REGION

REGION Network 23: LIFE BIT ALARM
   RUNG wire#powerrail
      I_Contact( "M_ONE" )
      wire#w1
      Contact( "M_0.5_SEC_2HZ" )
      { S7_Templates := "value_type := Int" } "DB7300_INTERLOCK_GENERAL".AUX_SIGNALS_INTERFACE.POWDER_PLC."LIFE SING COUNTER".CTU(r := "DB7300_INTERLOCK_GENERAL".POWDER_PLC.GENERAL.LIFE_BIT, pv := 0, cv => #COUNT_FOR_ERROR)
      Contact( "DB7300_INTERLOCK_GENERAL".POWDER_PLC.GENERAL.LIFE_BIT )
      R_Coil( "DB7300_INTERLOCK_GENERAL".POWDER_PLC.GENERAL.LIFE_BIT )
   END_RUNG
   RUNG wire#w1
      { S7_Templates := "SrcType := Int" } GE_Contact(in1 := #COUNT_FOR_ERROR, in2 := 4)
      I_Contact( "DB2031_CYCLES_GENERAL".MANUAL_LOAD_CYCLE.CYCLE_SELECTED )
      wire#w2
      Contact( "DB2120_MPP_ITC_IPC".MACHINE_ON_DELAYED )
      Contact( "M_DUMMY_OFF" )
      wire#w3
      Coil( "DB7300_INTERLOCK_GENERAL".AUX_SIGNALS_INTERFACE.POWDER_PLC.LIFE_BIT_FAULT )
   END_RUNG
   RUNG wire#w1
      Contact( "DB7300_INTERLOCK_GENERAL".AUX_SIGNALS_INTERFACE.POWDER_PLC.LIFE_BIT_FAULT )
      I_Contact( "DB2120_MPP_ITC_IPC".RESET_FAULTS )
   END_RUNG wire#w2
   RUNG wire#w3
      Coil( "DB426_ALARMS_WARNINGS".GENERAL."704410" )
   END_RUNG
   // the same network as SCL:
   "DB7300_INTERLOCK_GENERAL".AUX_SIGNALS_INTERFACE.POWDER_PLC."LIFE SING COUNTER".CTU(CU := NOT "M_ONE" AND "M_0.5_SEC_2HZ",
                           R := "DB7300_INTERLOCK_GENERAL".POWDER_PLC.GENERAL.LIFE_BIT,
                           PV := 0,
                           CV => #COUNT_FOR_ERROR);
   IF "DB7300_INTERLOCK_GENERAL".AUX_SIGNALS_INTERFACE.POWDER_PLC."LIFE SING COUNTER".Q AND "DB7300_INTERLOCK_GENERAL".POWDER_PLC.GENERAL.LIFE_BIT THEN
       "DB7300_INTERLOCK_GENERAL".POWDER_PLC.GENERAL.LIFE_BIT := FALSE;
   END_IF;
   "DB7300_INTERLOCK_GENERAL".AUX_SIGNALS_INTERFACE.POWDER_PLC.LIFE_BIT_FAULT := NOT "M_ONE" AND (((#COUNT_FOR_ERROR >= 4) AND NOT "DB2031_CYCLES_GENERAL".MANUAL_LOAD_CYCLE.CYCLE_SELECTED) OR ("DB7300_INTERLOCK_GENERAL".AUX_SIGNALS_INTERFACE.POWDER_PLC.LIFE_BIT_FAULT AND NOT "DB2120_MPP_ITC_IPC".RESET_FAULTS)) AND "DB2120_MPP_ITC_IPC".MACHINE_ON_DELAYED AND "M_DUMMY_OFF";
   "DB426_ALARMS_WARNINGS".GENERAL."704410" := "DB7300_INTERLOCK_GENERAL".AUX_SIGNALS_INTERFACE.POWDER_PLC.LIFE_BIT_FAULT;
END_REGION

REGION Network 24: IMMEDIATE STOP AND STOP END OF CYCLE ALARMS
   RUNG wire#powerrail
      I_Contact( "DB7300_INTERLOCK_GENERAL".AUX_SIGNALS_INTERFACE.POWDER_PLC.LIFE_BIT_FAULT )
      Not()
      Move(in := #FC_NUMBER, out1 => "DB440_MACHINE_ALARM_DECODING".GLOBAL_ALARMS_MACHINE.ALARM_DECODING)
      S_Coil( "DB440_MACHINE_ALARM_DECODING".ALARMS_CENTRAL.IS_ALARMS )
   END_RUNG
   // the same network as SCL:
   IF NOT (NOT "DB7300_INTERLOCK_GENERAL".AUX_SIGNALS_INTERFACE.POWDER_PLC.LIFE_BIT_FAULT) THEN
       "DB440_MACHINE_ALARM_DECODING".GLOBAL_ALARMS_MACHINE.ALARM_DECODING := #FC_NUMBER;
       "DB440_MACHINE_ALARM_DECODING".ALARMS_CENTRAL.IS_ALARMS := TRUE;
   END_IF;
END_REGION
END_FUNCTION
